(* IEC 61131-3 sources: plc-home-automation/home_automation/lighting_heating_updated/src/persist, 3 files *)

(* ---- PersistGlobals.st ---- *)
VAR_GLOBAL CONSTANT
    C_REALS_TO_PERSIST : INT      := C_HEATING_ZONES + 11;
    C_BOOLS_TO_PERSIST : INT      := 9;
    C_INTS_TO_PERSIST  : INT      := 2;
    C_TIMES_TO_PERSIST : INT      := 8;

    C_PERSIST_DIRECTORY_ROOT : STRING           := 'PST';
    C_PERSIST_HEATING_IPID_SUBDIR : STRING      := '';
    C_PERSIST_HEATING_SUBDIR : STRING           := '/HEATING';
    C_PERSIST_ROOM_TEMPERATURE_SUBDIR : STRING  := '/TEMP';
    C_PERSIST_BOILER_CONTROL_SUBDIR : STRING    := '/BOILER';
    C_VENTILLATION_SUBDIR : STRING              := '/VENT';
    C_WATERING_SUBDIR : STRING                  := '/WATER';
    C_UTILS_SUBDIR : STRING                     := '/UTILS';
END_VAR

VAR_GLOBAL
    REALS_TO_PERSIST : ARRAY [1 .. C_REALS_TO_PERSIST] OF PTR_TO REAL;
    REALS_TO_PERSIST_DIRS : ARRAY [1 .. C_REALS_TO_PERSIST] OF STRING;
    REALS_TO_PERSIST_NAMES : ARRAY [1 .. C_REALS_TO_PERSIST] OF STRING;

    BOOLS_TO_PERSIST : ARRAY [1 .. C_BOOLS_TO_PERSIST] OF PTR_TO BOOL;
    BOOLS_TO_PERSIST_DIRS : ARRAY [1 .. C_BOOLS_TO_PERSIST] OF STRING;
    BOOLS_TO_PERSIST_NAMES : ARRAY [1 .. C_BOOLS_TO_PERSIST] OF STRING;

    INTS_TO_PERSIST : ARRAY [1 .. C_INTS_TO_PERSIST] OF PTR_TO INT;
    INTS_TO_PERSIST_DIRS : ARRAY [1 .. C_INTS_TO_PERSIST] OF STRING;
    INTS_TO_PERSIST_NAMES : ARRAY [1 .. C_INTS_TO_PERSIST] OF STRING;

    TIMES_TO_PERSIST : ARRAY [1 .. C_TIMES_TO_PERSIST] OF PTR_TO TIME;
    TIMES_TO_PERSIST_DIRS : ARRAY [1 .. C_TIMES_TO_PERSIST] OF STRING;
    TIMES_TO_PERSIST_NAMES : ARRAY [1 .. C_TIMES_TO_PERSIST] OF STRING;

END_VAR

(* ---- Persist.st ---- *)
PROGRAM PersistData
  VAR_INPUT
  END_VAR
  VAR_OUTPUT
  END_VAR
  VAR
    init : BOOL := FALSE;
    realPersistors : ARRAY [1 .. C_REALS_TO_PERSIST] OF PersistReal;
    boolPersistors : ARRAY [1 .. C_BOOLS_TO_PERSIST] OF PersistBool;
    intPersistors : ARRAY  [1 .. C_INTS_TO_PERSIST]  OF PersistInt;
    timePersistors : ARRAY [1 .. C_TIMES_TO_PERSIST] OF PersistTime;

    i: INT := 0;
  END_VAR
  VAR_TEMP
  END_VAR

  FOR i := 1 to C_REALS_TO_PERSIST DO
    realPersistors[i](compilerBugPlaceholder := init,
      variableToPersist := REALS_TO_PERSIST[i]^,
      dirPath := REALS_TO_PERSIST_DIRS[i],
      fileName := REALS_TO_PERSIST_NAMES[i],
      toWrite := init);
  END_FOR;

  FOR i := 1 to C_BOOLS_TO_PERSIST DO
    boolPersistors[i](compilerBugPlaceholder := init,
      variableToPersist := BOOLS_TO_PERSIST[i]^,
      dirPath := BOOLS_TO_PERSIST_DIRS[i],
      fileName := BOOLS_TO_PERSIST_NAMES[i],
      toWrite := init);
  END_FOR;

  FOR i := 1 to C_INTS_TO_PERSIST DO
    intPersistors[i](compilerBugPlaceholder := init,
      variableToPersist := INTS_TO_PERSIST[i]^,
      dirPath := INTS_TO_PERSIST_DIRS[i],
      fileName := INTS_TO_PERSIST_NAMES[i],
      toWrite := init);
  END_FOR;

  FOR i := 1 to C_TIMES_TO_PERSIST DO
    timePersistors[i](compilerBugPlaceholder := init,
      variableToPersist := TIMES_TO_PERSIST[i]^,
      dirPath := TIMES_TO_PERSIST_DIRS[i],
      fileName := TIMES_TO_PERSIST_NAMES[i],
      toWrite := init);
  END_FOR;

  init := TRUE;

END_PROGRAM

(* ---- PersistInit.st ---- *)
PROGRAM PersistInit
  VAR_INPUT
  END_VAR
  VAR_OUTPUT
  END_VAR
  VAR
    init : BOOL := FALSE;
    i : INT := 0;
    ipidPath : STRING;
    heatingRootPath : STRING;
    roomTempPath : STRING;
    boilerControlPath : STRING;
    ventillationControlPath : STRING;
    wateringControlPath : STRING;
    utilsControlPath : STRING;
  END_VAR
  VAR_TEMP
  END_VAR

  ipidPath := CONCAT(C_PERSIST_DIRECTORY_ROOT, C_PERSIST_HEATING_IPID_SUBDIR);
  heatingRootPath := CONCAT(C_PERSIST_DIRECTORY_ROOT, C_PERSIST_HEATING_SUBDIR);
  roomTempPath := CONCAT(heatingRootPath, C_PERSIST_ROOM_TEMPERATURE_SUBDIR);
  boilerControlPath := CONCAT(heatingRootPath, C_PERSIST_BOILER_CONTROL_SUBDIR);
  ventillationControlPath := CONCAT(C_PERSIST_DIRECTORY_ROOT, C_VENTILLATION_SUBDIR);
  wateringControlPath := CONCAT(C_PERSIST_DIRECTORY_ROOT, C_WATERING_SUBDIR);
  utilsControlPath := CONCAT(C_PERSIST_DIRECTORY_ROOT, C_UTILS_SUBDIR);

  createDirectory(dirPath := C_PERSIST_DIRECTORY_ROOT);
    createDirectory(dirPath := ipidPath);
    createDirectory(dirPath := heatingRootPath);
        createDirectory(dirPath := roomTempPath);
        createDirectory(dirPath := boilerControlPath);
    createDirectory(dirPath := ventillationControlPath);
    createDirectory(dirPath := wateringControlPath);

  IF NOT init THEN
    FOR i := 1 TO C_HEATING_ZONES DO
      REALS_TO_PERSIST[i] := DESIRED_TEMPERATURES[i-1];
      REALS_TO_PERSIST_NAMES[i] := INT_TO_STRING(i);
      REALS_TO_PERSIST_DIRS[i] := roomTempPath;
    END_FOR;

    REALS_TO_PERSIST[C_HEATING_ZONES + 1]        := ADR(IPID_K);
    REALS_TO_PERSIST_NAMES[C_HEATING_ZONES + 1]  := 'IPIDK';
    REALS_TO_PERSIST_DIRS[C_HEATING_ZONES + 1]   := boilerControlPath;
    REALS_TO_PERSIST[C_HEATING_ZONES + 2]        := ADR(IPID_TD);
    REALS_TO_PERSIST_NAMES[C_HEATING_ZONES + 2]  := 'IPIDTD';
    REALS_TO_PERSIST_DIRS[C_HEATING_ZONES + 2]   := boilerControlPath;
    REALS_TO_PERSIST[C_HEATING_ZONES + 3]        := ADR(IPID_TI);
    REALS_TO_PERSIST_NAMES[C_HEATING_ZONES + 3]  := 'IPIDTI';
    REALS_TO_PERSIST_DIRS[C_HEATING_ZONES + 3]   := boilerControlPath;
    REALS_TO_PERSIST[C_HEATING_ZONES + 4]        := ADR(OVERSHOOT_HISTERESIS);
    REALS_TO_PERSIST_NAMES[C_HEATING_ZONES + 4]  := 'OVHISTER';
    REALS_TO_PERSIST_DIRS[C_HEATING_ZONES + 4]   := boilerControlPath;

    REALS_TO_PERSIST[C_HEATING_ZONES + 5]        := ADR(HOT_WATER_TEMPERATURE);
    REALS_TO_PERSIST_NAMES[C_HEATING_ZONES + 5]  := 'HOTWTEMP';
    REALS_TO_PERSIST_DIRS[C_HEATING_ZONES + 5]   := boilerControlPath;

    REALS_TO_PERSIST[C_HEATING_ZONES + 6]        := ADR(WATERING_CUTOFF_TEMPERATURE);
    REALS_TO_PERSIST_NAMES[C_HEATING_ZONES + 6]  := 'WATTEMP';
    REALS_TO_PERSIST_DIRS[C_HEATING_ZONES + 6]   := wateringControlPath;
    REALS_TO_PERSIST[C_HEATING_ZONES + 7]        := ADR(FRONT_GRASS_WATERING_OFFSET);
    REALS_TO_PERSIST_NAMES[C_HEATING_ZONES + 7]  := 'FGOFFSET';
    REALS_TO_PERSIST_DIRS[C_HEATING_ZONES + 7]   := wateringControlPath;
    REALS_TO_PERSIST[C_HEATING_ZONES + 8]        := ADR(REAR_GRASS_WATERING_OFFSET);
    REALS_TO_PERSIST_NAMES[C_HEATING_ZONES + 8]  := 'RGOFFSET';
    REALS_TO_PERSIST_DIRS[C_HEATING_ZONES + 8]   := wateringControlPath;
    REALS_TO_PERSIST[C_HEATING_ZONES + 9]        := ADR(FRONT_GRASS_WATERING_TEMPERATURE_COEFFICIENT);
    REALS_TO_PERSIST_NAMES[C_HEATING_ZONES + 9]  := 'FGCOEFF';
    REALS_TO_PERSIST_DIRS[C_HEATING_ZONES + 9]   := wateringControlPath;
    REALS_TO_PERSIST[C_HEATING_ZONES + 10]       := ADR(REAR_GRASS_WATERING_TEMPERATURE_COEFFICIENT);
    REALS_TO_PERSIST_NAMES[C_HEATING_ZONES + 10] := 'RGCOEFF';
    REALS_TO_PERSIST_DIRS[C_HEATING_ZONES + 10]  := wateringControlPath;

    REALS_TO_PERSIST[C_HEATING_ZONES + 11]       := ADR(EXTERNAL_AVERAGE_TEMPERATURE);
    REALS_TO_PERSIST_NAMES[C_HEATING_ZONES + 11] := 'EXTAVGTEMP';
    REALS_TO_PERSIST_DIRS[C_HEATING_ZONES + 11]  := utilsControlPath;

    BOOLS_TO_PERSIST[1]       := ADR(HEATING_ENABLE);
    BOOLS_TO_PERSIST_NAMES[1] := 'BOILER';
    BOOLS_TO_PERSIST_DIRS[1]  := boilerControlPath;
    BOOLS_TO_PERSIST[2]       := ADR(HOT_WATER_ENABLE);
    BOOLS_TO_PERSIST_DIRS[2]  := boilerControlPath;
    BOOLS_TO_PERSIST_NAMES[2] := 'HOTWATER';
    BOOLS_TO_PERSIST[3]       := ADR(PRESENCE_BASED_HEATING_CONTROL);
    BOOLS_TO_PERSIST_NAMES[3] := 'BOILERPC';
    BOOLS_TO_PERSIST_DIRS[3]  := boilerControlPath;
    BOOLS_TO_PERSIST[4]       := ADR(PRESENCE_BASED_HOT_WATER_CONTROL);
    BOOLS_TO_PERSIST_DIRS[4]  := boilerControlPath;
    BOOLS_TO_PERSIST_NAMES[4] := 'HOTWPC';
    BOOLS_TO_PERSIST[5]       := ADR(PRESENCE_BASED_VENTILLATION_CONTROL);
    BOOLS_TO_PERSIST_DIRS[5]  := ventillationControlPath;
    BOOLS_TO_PERSIST_NAMES[5] := 'VENTPC';
    BOOLS_TO_PERSIST[6]       := ADR(COOLING_PRIORITY_VENTILLATION_CONTROL);
    BOOLS_TO_PERSIST_DIRS[6]  := ventillationControlPath;
    BOOLS_TO_PERSIST_NAMES[6] := 'VENTCC';
    //
    BOOLS_TO_PERSIST[7]       := ADR(WATERING_ENABLE);
    BOOLS_TO_PERSIST_DIRS[7]  := wateringControlPath;
    BOOLS_TO_PERSIST_NAMES[7] := 'WATON';
    BOOLS_TO_PERSIST[8]       := ADR(TEMPERATURE_BASED_WATERING_CONTROL);
    BOOLS_TO_PERSIST_DIRS[8]  := wateringControlPath;
    BOOLS_TO_PERSIST_NAMES[8] := 'RAINON';
    BOOLS_TO_PERSIST[9]       := ADR(RAIN_BASED_WATERING_CONTROL);
    BOOLS_TO_PERSIST_DIRS[9]  := wateringControlPath;
    BOOLS_TO_PERSIST_NAMES[9] := 'TEMPON';

    INTS_TO_PERSIST[1]        := ADR(NILAN_DESIRED_VENTILLATION_LEVEL);
    INTS_TO_PERSIST_DIRS[1]   := ventillationControlPath;
    INTS_TO_PERSIST_NAMES[1]  := 'FANLEVEL';
    INTS_TO_PERSIST[2]        := ADR(NILAN_DESIRED_TEMPERATURE);
    INTS_TO_PERSIST_DIRS[2]   := ventillationControlPath;
    INTS_TO_PERSIST_NAMES[2]  := 'VENTTEMP';

    TIMES_TO_PERSIST[1]        := ADR(WATERING_START_TIME[1]);
    TIMES_TO_PERSIST_DIRS[1]   := wateringControlPath;
    TIMES_TO_PERSIST_NAMES[1]  := 'START1';
    TIMES_TO_PERSIST[2]        := ADR(FRONT_GRASS_WATERING_TIME[1]);
    TIMES_TO_PERSIST_DIRS[2]   := wateringControlPath;
    TIMES_TO_PERSIST_NAMES[2]  := 'FRONT1';
    TIMES_TO_PERSIST[3]        := ADR(REAR_GRASS_WATERING_TIME[1]);
    TIMES_TO_PERSIST_DIRS[3]   := wateringControlPath;
    TIMES_TO_PERSIST_NAMES[3]  := 'REAR1';
    TIMES_TO_PERSIST[4]        := ADR(BUSHES_WATERING_TIME[1]);
    TIMES_TO_PERSIST_DIRS[4]   := wateringControlPath;
    TIMES_TO_PERSIST_NAMES[4]  := 'BUSH1';
    TIMES_TO_PERSIST[5]        := ADR(WATERING_START_TIME[2]);
    TIMES_TO_PERSIST_DIRS[5]   := wateringControlPath;
    TIMES_TO_PERSIST_NAMES[5]  := 'START2';
    TIMES_TO_PERSIST[6]        := ADR(FRONT_GRASS_WATERING_TIME[2]);
    TIMES_TO_PERSIST_DIRS[6]   := wateringControlPath;
    TIMES_TO_PERSIST_NAMES[6]  := 'FRONT2';
    TIMES_TO_PERSIST[7]        := ADR(REAR_GRASS_WATERING_TIME[2]);
    TIMES_TO_PERSIST_DIRS[7]   := wateringControlPath;
    TIMES_TO_PERSIST_NAMES[7]  := 'REAR2';
    TIMES_TO_PERSIST[8]        := ADR(BUSHES_WATERING_TIME[2]);
    TIMES_TO_PERSIST_DIRS[8]   := wateringControlPath;
    TIMES_TO_PERSIST_NAMES[8]  := 'BUSH2';

    init := TRUE;

  ELSE
    // No operation
  END_IF;

END_PROGRAM
